// TIA Portal V16 export
// export: Created 2024-12-03T15:41:46.517708Z, ExportSetting WithReadOnly, DisplayName Totally Integrated Automation Portal, DisplayVersion V16 Update 6, DisplayName TIA Portal Version Control Interface, DisplayVersion V16 Update 2, DisplayName TIA Portal Openness, DisplayVersion V16 Update 6, DisplayName TIA Portal Teamcenter Gateway, DisplayVersion V16, DisplayName SINAMICS Startdrive Advanced, DisplayVersion V16 Update 5, DisplayName SINAMICS Startdrive G130, G150, S120, S150, SINAMICS MV, S210, DisplayVersion V16 Update 5, DisplayName SINAMICS Startdrive G110M, G120, G120C, G120D, G120P, G115D, DisplayVersion V16 Update 5, DisplayName STEP 7 Professional, DisplayVersion V16 Update 6, DisplayName STEP 7 Safety, DisplayVersion V16, DisplayName WinCC Advanced / Unified PC, DisplayVersion V16 Update 6
TYPE "WRITE_POINT_UDT"
// stored: CreationDate 2022-04-18T07:34:22.161404Z, InterfaceModifiedDate 2022-04-18T07:34:26.4021311Z, IsConsistent true, LibraryConformanceStatus The object is library-conformant., ModifiedDate 2022-04-18T07:34:26.4021311Z
   STRUCT
      I_Measurement : String[50];
      I_tags : String;
      I_fields : String;
      I_time : String[30];
   END_STRUCT;
END_TYPE
